INTERFACE I_Curtain

METHOD Close : BOOL
VAR_INPUT
	IN: BOOL;
END_VAR
END_METHOD

METHOD Open : BOOL
VAR_INPUT
	IN: BOOL;
END_VAR
END_METHOD

END_INTERFACE

(* stored: Version 1.1.0.1, ProductVersion 3.1.4024.13
   Itf I_Curtain: Id {afa632ab-a7d5-40fd-a66c-55f2d42c27f7}
   Method Close: Id {d0e0b6fe-adef-401c-a4f7-6f6a16aa06bf}
   Method Open: Id {ea343dad-57ad-46dd-b91f-59c666ee1946} *)
